Staubli VAL3: GotoPosition.pgx

program GotoPosition(num& arrayValue[])
  local num result
begin
  //*******************************************************************************
  //*   ______
  //*  / _____) /|
  //* | |      / /
  //* | | /\  / /
  //* | | \ \/ /  _      Copyright (c) KEOLABS, 2016
  //* | |  \__/  | |        http://www.keolabs.com
  //* | |________| |
  //*  \__________/
  //*
  //********************************************************************************
  //*@file          : GotoPosition
  //*@author        : Yves Ragot
  //*@version       : $Id: GotoPosition.pgx 1198 2016-10-07 06:48:14Z yves $
  //*@brief         : GotoPosition command treatment (absolute Cartesian mouvement)
  //*
  //*******************************************************************************/

  // get target point
  pTargetPoint.trsf.x = arrayValue[0]
  pTargetPoint.trsf.y = arrayValue[1]
  pTargetPoint.trsf.z = arrayValue[2]
  pTargetPoint.trsf.rx = arrayValue[3]
  pTargetPoint.trsf.ry = arrayValue[4]
  pTargetPoint.trsf.rz = arrayValue[5]

  CartesianMode = true

  // launch mouvement
  ExecuteMotion = true

  // wait for end of execution
  wait(ExecuteMotion == false)

end
